{attribute 'strict'}
{attribute 'to_string'}
TYPE XTSMainState_enum : (
        MS_DISABLED					:= 0,
        MS_INITIALIZING_MOVERS		:= 10,
		MS_ONESHOT_ENABLE			:= 20,
        MS_ENABLING_MOVERS			:= 30,
        MS_INITIALIZING_OBJECTIVES	:= 40,
		MS_ACTIVATE_TRACKS			:= 45,
		MS_WAIT_FOR_TRACKS			:= 46,
        MS_ENABLED					:= 50,
		MS_STARTUP					:= 51,
        MS_RUN						:= 60,
		MS_ONESHOT_STOP				:= 70,
        MS_STOPPING					:= 80,
        MS_STOPPED					:= 90,
		MS_ONESHOT_DISABLE			:= 100,
        MS_DISABLING				:= 110,
        MS_ERROR					:= 120,
        MS_DEBUG					:= 1000
    );
END_TYPE

(* stored: Version 1.1.0.1, ProductVersion 3.1.4024.12
   DUT XTSMainState_enum: Id {9ee55b6c-1c5f-06af-2bfa-dd4834005e9d} *)
